INTERFACE IAnalogueInput

PROPERTY Error : bool
GET
END_GET
END_PROPERTY

METHOD GetConvertedValue : REAL
VAR_INPUT
END_VAR
END_METHOD

METHOD GetRawValue : int
VAR_INPUT
END_VAR
END_METHOD

END_INTERFACE

(* stored: Version 1.1.0.1, ProductVersion 3.1.4024.5
   Itf IAnalogueInput: Id {e636cff6-7a32-4dc7-89f1-d79afca9588b}
   Property Error: Id {ceb3dd31-0f47-4b83-8621-f22886152bee}
   Get Get: Id {d8504d6a-40d2-406d-b6b7-8e5d4a91f722}
   Method GetConvertedValue: Id {89754de7-153c-4a85-9bd0-ede4a8f0cc1d}
   Method GetRawValue: Id {8d200988-97d3-474f-bb0a-ffaada991048} *)
